PROGRAM YAHOO_WEATHER_DEMO_1
VAR
	IP_C: IP_C;
	S_BUF: NETWORK_BUFFER;
	R_BUF: NETWORK_BUFFER;
	IP_CONTROL_1: IP_CONTROL;
	activate: BOOL;
	done: BOOL;
	busy: BOOL;
	error_c: DWORD;
	error_t: BYTE;
	YAHOO_WEATHER: YAHOO_WEATHER;
	YW_DATA: YAHOO_WEATHER_DATA;
	CLK_PRG: CLK_PRG;
	YAHOO_WEATHER_DESC_GE: YAHOO_WEATHER_DESC_GE;
	YAHOO_WEATHER_ICON_OSCAT: YAHOO_WEATHER_ICON_OSCAT;
END_VAR
VAR // added by the converter: edge detectors and wires of the graphical bodies
    _w1 : ANY;
END_VAR

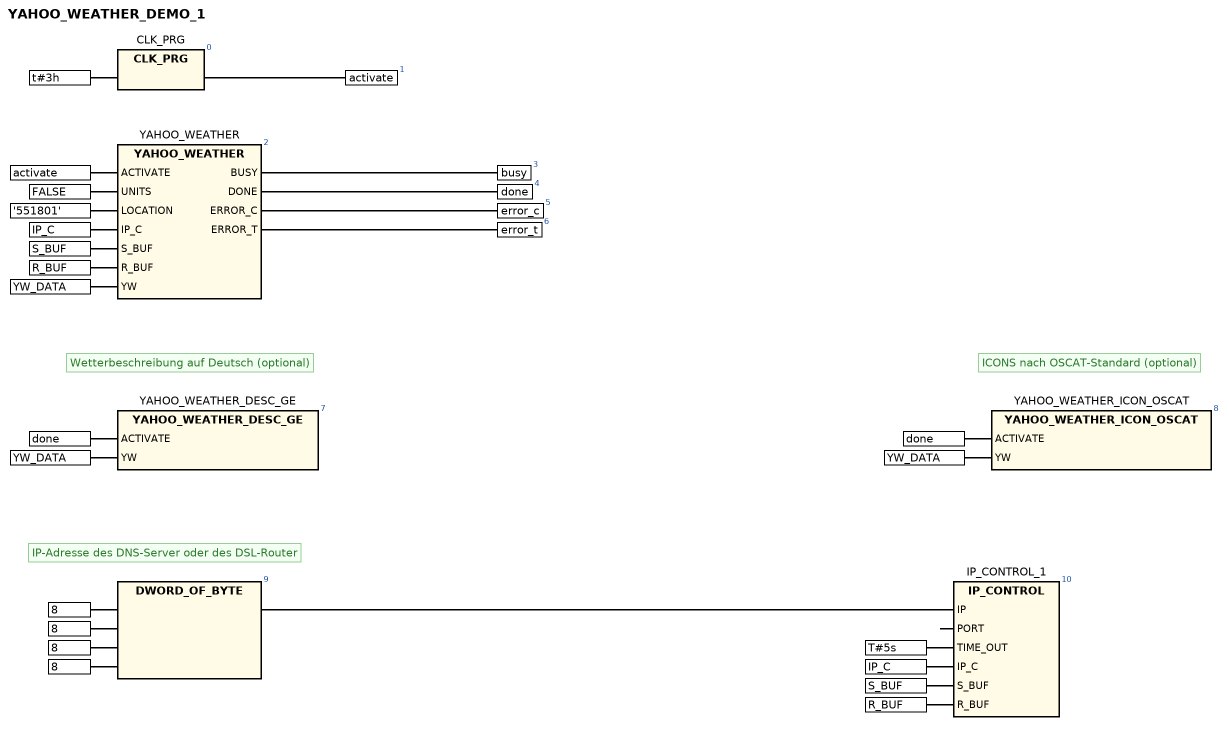
CLK_PRG(_in1 := t#3h);
activate := CLK_PRG._out1;
YAHOO_WEATHER(
    ACTIVATE := activate,
    UNITS := FALSE,
    LOCATION := '551801',
    IP_C := IP_C,
    S_BUF := S_BUF,
    R_BUF := R_BUF,
    YW := YW_DATA);
busy := YAHOO_WEATHER.BUSY;
done := YAHOO_WEATHER.DONE;
error_c := YAHOO_WEATHER.ERROR_C;
error_t := YAHOO_WEATHER.ERROR_T;
// Wetterbeschreibung auf Deutsch (optional)
YAHOO_WEATHER_DESC_GE(ACTIVATE := done, YW := YW_DATA);
// ICONS nach OSCAT-Standard (optional)
YAHOO_WEATHER_ICON_OSCAT(ACTIVATE := done, YW := YW_DATA);
// IP-Adresse des DNS-Server oder des DSL-Router
_w1 := DWORD_OF_BYTE(8, 8, 8, 8);
IP_CONTROL_1(IP := _w1, TIME_OUT := T#5s, IP_C := IP_C, S_BUF := S_BUF, R_BUF := R_BUF); // IP_CONTROL

END_PROGRAM

(* stored: Version 1.1.0.1, ProductVersion 3.1.4024.0
   POU YAHOO_WEATHER_DEMO_1: Id {1efc18a4-c3a8-4419-9bb9-a7658f0543fe}, SpecialFunc None *)
